TYPE ST_ChannelConfig :
STRUCT
	sName : STRING(255);
	eDataType : E_ChannelDataType;
	sDescription : STRING(255);
	sUnit : STRING(255);
	aEnumTypes : ARRAY[0..SiftClientParameters.MAX_NUM_ENUMS_PER_CHANNEL - 1] OF ST_EnumType;
	nNumEnumTypes : UDINT;
	
	Value : _U_SiftChannelValue;
END_STRUCT
END_TYPE

(* stored: Version 1.1.0.1
   DUT ST_ChannelConfig: Id {fa8bf50b-664e-4788-a759-59b3e531d27f} *)
